PROGRAM PRG_Compilation
VAR
	fbButton		: FB_HMIEButton;
	fbButtonHMI		: FB_HMIEButton_HMI (itfButton := fbButton);
	fbMenu			: FB_HMIEMenu;
	fbMenuHMI		: FB_HMIEMenu_HMI (itfMenu := fbMenu);
END_VAR

END_PROGRAM

(* stored: Version 1.1.0.1
   POU PRG_Compilation: Id {c5cc7d45-cf9d-4ea0-97cb-d3fd07051ddf}, SpecialFunc None *)
